{attribute addProperty BoxType "EK1122-0000-0018"}
{attribute addProperty Id "Beckhoff_EP8xxxsub_EK1100EK1100_179A0949162A_0001_EP8309_0022_0021EP8309_4876315539449.25A_0002_EP8309_1022_0016EP8309_4876315539449.25A_0003_EP8309_1022_0017EP8309_4876315539449.25A_0004_EP8309_1022_0018EP8309_4876315539449.25"}
{attribute addProperty CRC "151154005"}
{attribute addProperty SizeInBites "1592"}
{attribute addProperty SizeInBytes "199"}
TYPE Beckhoff_EP8xxxEK1122_09026D55 EXTENDS EK1122_179A0949 :
STRUCT
	{attribute addProperty Name "Beckhoff_EP8xxxsub_EK1100"}
	Beckhoff_EP8xxxsub_EK1100 : EK1100_179A0949;
	{attribute addProperty Name "A_0001_EP8309_0022_0021"}
	A_0001_EP8309_0022_0021 : EP8309_48763155;
	{attribute addProperty Name "A_0002_EP8309_1022_0016"}
	A_0002_EP8309_1022_0016 : EP8309_48763155;
	{attribute addProperty Name "A_0003_EP8309_1022_0017"}
	A_0003_EP8309_1022_0017 : EP8309_48763155;
	{attribute addProperty Name "A_0004_EP8309_1022_0018"}
	A_0004_EP8309_1022_0018 : EP8309_48763155;
END_STRUCT
END_TYPE

(* stored: Version 1.2.0.0, ProductVersion 3.1.4024.9
   DUT Beckhoff_EP8xxxEK1122_09026D55: Id {925a8b3e-1ac9-41be-aca9-0ad69ec70b29} *)
